FUNCTION_BLOCK AE_AX_AX_SPLIT (* AE_AX passthrough (Socket to Plug) plus an extra AX Plug mirroring the AE_AX backward (state) channel *)
  (* Standard: 61499-2; Function: Any Event coming in by IN is forwarded to OUT unchanged; the backward Event/Bool fired into OUT by the downstream Socket is relayed both back through IN and out via AX_OUT; Description: Copyright (c) 2026 HR Agrartechnik GmbH This program and the accompanying materials are made available under the terms of the Eclipse Public License 2.0 which is available at https://www.eclipse.org/legal/epl-2.0/ SPDX-License-Identifier: EPL-2.0 *)
  (* Version 1.0, 2026-09-03, Franz Höpfinger, HR Agrartechnik GmbH, Initial Version *)
  PACKAGE adapter::events::bidirectional;
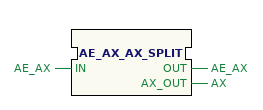
  SOCKETS
    IN : adapter::types::bidirectional::AE_AX; (* Input *)
  END_SOCKETS
  PLUGS
    OUT : adapter::types::bidirectional::AE_AX; (* Output *)
    AX_OUT : adapter::types::unidirectional::AX; (* mirrors the AE_AX backward (state) channel *)
  END_PLUGS
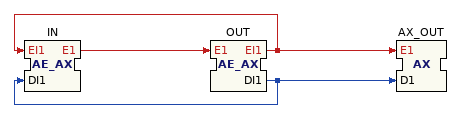
  EVENT_CONNECTIONS
    IN.E1 TO OUT.E1;
    OUT.EI1 TO IN.EI1;
    OUT.EI1 TO AX_OUT.E1;
  END_CONNECTIONS
  DATA_CONNECTIONS
    OUT.DI1 TO IN.DI1;
    OUT.DI1 TO AX_OUT.D1;
  END_CONNECTIONS
END_FUNCTION_BLOCK
